Fanuc TP program (LS listing): UP022.LS

/PROG  UP022
/ATTR
OWNER		= MNEDITOR;
COMMENT		= "Soldadura Est.";
PROG_SIZE	= 14814;
CREATE		= DATE 23-07-08  TIME 22:43:52;
MODIFIED	= DATE 24-03-28  TIME 23:41:50;
FILE_NAME	= UP002;
VERSION		= 0;
LINE_COUNT	= 64;
MEMORY_SIZE	= 27222;
PROTECT		= READ_WRITE;
TCD:  STACK_SIZE	= 500,
      TASK_PRIORITY	= 50,
      TIME_SLICE	= 0,
      BUSY_LAMP_OFF	= 0,
      ABORT_REQUEST	= 0,
      PAUSE_REQUEST	= 0;
DEFAULT_GROUP	= 1,1,1,1,*;
CONTROL_CODE	= 00000001 00000000;
/APPL
/MN
   1:  UFRAME_NUM=1 ;
   2:  UTOOL_NUM=2 ;
   3:  PAYLOAD[2] ;
   4:J P[1] 100% CNT0 ACC100 TB    .10sec,P-SPS    ;
      1:  TC_ONLINE (ON) ;
      2:  DO[23]=OFF ;
      3:  TIMER[4]=RESET ;
      4:  TIMER[4]=START ;
      5:  CALL MAKRO050    ;
      6:  !Lib. de Herramientas ;
      7:  DO[80]=ON ;
      8:  DO[79]=ON ;
      9:  DO[78]=OFF ;
     10:  DO[77]=OFF ;
     11:  DO[76]=OFF ;
     12:  DO[75]=ON ;
     13:  DO[73]=OFF ;
     14:  !RLib. de Anticolisiones ;
     15:  DO[41]=ON ;
     16:  DO[42]=ON ;
     17:  DO[43]=ON ;
     18:  DO[44]=ON ;
     19:  DO[45]=ON ;
     20:  DO[46]=ON ;
     21:  !Apagar Pos. Base ;
     22:  DO[15]=OFF ;
     23:  !Robot en Trayectoria ;
     24:  DO[16]=ON ;
     25:  !Basculante en Pos. de Reposo ;
     26:  IF (!DI[842] AND DO[12]),CALL MAKRO072 ;
     27:  WAIT (M[96])    ;
     28:  WAIT (DI[23])    ;
     29:  DO[23]=(ON) ;
     30:  TC_ONLINE (M[1] AND M[30] AND M[31] AND M[34] AND M[95] AND M[96]) ;
       ------ ;
   5:J P[2] 100% CNT100 ACC100 TB   0.00sec,P-SPS    ;
      1:  TC_ONLINE (M[1] AND M[30] AND M[31] AND M[34] AND M[95] AND M[96]) ;
       ------ ;
   6:J P[3] 100% CNT100 ACC100 TB   0.00sec,P-SPS    ;
      1:  TC_ONLINE (M[1] AND M[30] AND M[31] AND M[34] AND M[95] AND M[96]) ;
       ------ ;
   7:J P[4] 100% CNT100 ACC100 TB   0.00sec,P-SPS    ;
      1:  TC_ONLINE (M[1] AND M[30] AND M[31] AND M[34] AND M[95] AND M[96]) ;
       ------ ;
   8:J P[5] 100% CNT100 ACC100 TB   0.00sec,P-SPS    ;
      1:  TC_ONLINE (M[1] AND M[30] AND M[31] AND M[34] AND M[95] AND M[96]) ;
       ------ ;
   9:  !5QA802035B_019_T_PS_0007 ;
  10:  !Punto de Sol. No. 10081 ;
  11:J P[6] 100% CNT0 ACC100 TB    .10sec,P-SPS Offset,PR[11]    ;
      1:  TC_ONLINE (ON) ;
      2:  DO[23]=OFF ;
      3:  WAIT (!DI[16] AND DI[23])    ;
      4:  CALL VW_USER(Basic1,EZSP,Nr1,ProgNr=99, , ,S-Punkt=10081,Fzg_Typ=7,EIN/AUS=ON) ;
      5:  GO[2]=(R[197]+20) ;
      6:  WAIT (!DI[129] OR DI[26])    ;
      7:  CALL MAKRO080    ;
      8:  WAIT (DI[23])    ;
      9:  DO[23]=ON ;
     10:  TC_ONLINE (M[1] AND M[30] AND M[31] AND M[34] AND M[95] AND M[96]) ;
       ------ ;
  12:J P[7] 100% CNT100 ACC100 TB   0.00sec,P-SPS    ;
      1:  TC_ONLINE (M[1] AND M[30] AND M[31] AND M[34] AND M[95] AND M[96]) ;
       ------ ;
  13:  !5QA802035B_019_T_PS_0008 ;
  14:  !Punto de Sol. No. 10082 ;
  15:J P[8] 100% CNT0 ACC100 TB    .10sec,P-SPS Offset,PR[11]    ;
      1:  TC_ONLINE (ON) ;
      2:  DO[23]=OFF ;
      3:  WAIT (!DI[16] AND DI[23])    ;
      4:  CALL VW_USER(Basic1,EZSP,Nr1,ProgNr=99, , ,S-Punkt=10082,Fzg_Typ=7,EIN/AUS=ON) ;
      5:  GO[2]=(R[197]+20) ;
      6:  WAIT (!DI[129] OR DI[26])    ;
      7:  CALL MAKRO080    ;
      8:  WAIT (DI[23])    ;
      9:  DO[23]=ON ;
     10:  TC_ONLINE (M[1] AND M[30] AND M[31] AND M[34] AND M[95] AND M[96]) ;
       ------ ;
  16:  !5QA802035B_019_T_PS_0002 ;
  17:  !Punto de Sol. No. 10083 ;
  18:J P[9] 100% CNT0 ACC100 TB    .10sec,P-SPS Offset,PR[11]    ;
      1:  TC_ONLINE (ON) ;
      2:  DO[23]=OFF ;
      3:  WAIT (!DI[16] AND DI[23])    ;
      4:  CALL VW_USER(Basic1,EZSP,Nr1,ProgNr=99, , ,S-Punkt=10083,Fzg_Typ=7,EIN/AUS=ON) ;
      5:  GO[2]=(R[197]+20) ;
      6:  WAIT (!DI[129] OR DI[26])    ;
      7:  CALL MAKRO080    ;
      8:  WAIT (DI[23])    ;
      9:  DO[23]=ON ;
     10:  TC_ONLINE (M[1] AND M[30] AND M[31] AND M[34] AND M[95] AND M[96]) ;
       ------ ;
  19:  !5QA802035B_019_T_PS_0003 ;
  20:  !Punto de Sol. No. 10084 ;
  21:J P[10] 100% CNT0 ACC100 TB    .10sec,P-SPS Offset,PR[11]    ;
      1:  TC_ONLINE (ON) ;
      2:  DO[23]=OFF ;
      3:  WAIT (!DI[16] AND DI[23])    ;
      4:  CALL VW_USER(Basic1,EZSP,Nr1,ProgNr=99, , ,S-Punkt=10084,Fzg_Typ=7,EIN/AUS=ON) ;
      5:  GO[2]=(R[197]+20) ;
      6:  WAIT (!DI[129] OR DI[26])    ;
      7:  CALL MAKRO080    ;
      8:  WAIT (DI[23])    ;
      9:  DO[23]=ON ;
     10:  TC_ONLINE (M[1] AND M[30] AND M[31] AND M[34] AND M[95] AND M[96]) ;
       ------ ;
  22:  !5QA802035B_019_T_PS_0009 ;
  23:  !Punto de Sol. No. 10085 ;
  24:J P[11] 100% CNT0 ACC100 TB    .10sec,P-SPS Offset,PR[11]    ;
      1:  TC_ONLINE (ON) ;
      2:  DO[23]=OFF ;
      3:  WAIT (!DI[16] AND DI[23])    ;
      4:  CALL VW_USER(Basic1,EZSP,Nr1,ProgNr=99, , ,S-Punkt=10085,Fzg_Typ=7,EIN/AUS=ON) ;
      5:  GO[2]=(R[197]+20) ;
      6:  WAIT (!DI[129] OR DI[26])    ;
      7:  CALL MAKRO080    ;
      8:  WAIT (DI[23])    ;
      9:  DO[23]=ON ;
     10:  TC_ONLINE (M[1] AND M[30] AND M[31] AND M[34] AND M[95] AND M[96]) ;
       ------ ;
  25:J P[12] 100% CNT100 ACC100 TB   0.00sec,P-SPS    ;
      1:  TC_ONLINE (M[1] AND M[30] AND M[31] AND M[34] AND M[95] AND M[96]) ;
       ------ ;
  26:   ;
  27:  !5QA802035B_019_T_PS_0001 ;
  28:  !Punto de Sol. No. 10086 ;
  29:J P[13] 100% CNT0 ACC100 TB    .10sec,P-SPS Offset,PR[11]    ;
      1:  TC_ONLINE (ON) ;
      2:  DO[23]=OFF ;
      3:  WAIT (!DI[16] AND DI[23])    ;
      4:  CALL VW_USER(Basic1,EZSP,Nr1,ProgNr=99, , ,S-Punkt=10086,Fzg_Typ=7,EIN/AUS=ON) ;
      5:  GO[2]=(R[197]+20) ;
      6:  WAIT (!DI[129] OR DI[26])    ;
      7:  CALL MAKRO080    ;
      8:  WAIT (DI[23])    ;
      9:  DO[23]=ON ;
     10:  TC_ONLINE (M[1] AND M[30] AND M[31] AND M[34] AND M[95] AND M[96]) ;
       ------ ;
  30:  !5QA802035B_019_T_PS_0004 ;
  31:  !Punto de Sol. No. 10087 ;
  32:J P[14] 100% CNT0 ACC100 TB    .10sec,P-SPS Offset,PR[11]    ;
      1:  TC_ONLINE (ON) ;
      2:  DO[23]=OFF ;
      3:  WAIT (!DI[16] AND DI[23])    ;
      4:  CALL VW_USER(Basic1,EZSP,Nr1,ProgNr=99, , ,S-Punkt=10087,Fzg_Typ=7,EIN/AUS=ON) ;
      5:  GO[2]=(R[197]+20) ;
      6:  WAIT (!DI[129] OR DI[26])    ;
      7:  CALL MAKRO080    ;
      8:  WAIT (DI[23])    ;
      9:  DO[23]=ON ;
     10:  TC_ONLINE (M[1] AND M[30] AND M[31] AND M[34] AND M[95] AND M[96]) ;
       ------ ;
  33:J P[15] 100% CNT100 ACC100 TB   0.00sec,P-SPS    ;
      1:  TC_ONLINE (M[1] AND M[30] AND M[31] AND M[34] AND M[95] AND M[96]) ;
       ------ ;
  34:  !5QA802035B_055_BN_PS_0001 ;
  35:  !Punto de Sol. No. 10088 ;
  36:J P[16] 100% CNT0 ACC100 TB    .10sec,P-SPS Offset,PR[11]    ;
      1:  TC_ONLINE (ON) ;
      2:  DO[23]=OFF ;
      3:  WAIT (!DI[16] AND DI[23])    ;
      4:  CALL VW_USER(Basic1,EZSP,Nr1,ProgNr=99, , ,S-Punkt=10088,Fzg_Typ=7,EIN/AUS=ON) ;
      5:  GO[2]=(R[197]+20) ;
      6:  WAIT (!DI[129] OR DI[26])    ;
      7:  CALL MAKRO080    ;
      8:  WAIT (DI[23])    ;
      9:  DO[23]=ON ;
     10:  TC_ONLINE (M[1] AND M[30] AND M[31] AND M[34] AND M[95] AND M[96]) ;
       ------ ;
  37:  !5QA802035B_019_T_PS_0005 ;
  38:  !Punto de Sol. No. 10089 ;
  39:J P[17] 100% CNT0 ACC100 TB    .10sec,P-SPS Offset,PR[11]    ;
      1:  TC_ONLINE (ON) ;
      2:  DO[23]=OFF ;
      3:  WAIT (!DI[16] AND DI[23])    ;
      4:  CALL VW_USER(Basic1,EZSP,Nr1,ProgNr=99, , ,S-Punkt=10089,Fzg_Typ=7,EIN/AUS=ON) ;
      5:  GO[2]=(R[197]+20) ;
      6:  WAIT (!DI[129] OR DI[26])    ;
      7:  CALL MAKRO080    ;
      8:  WAIT (DI[23])    ;
      9:  DO[23]=ON ;
     10:  TC_ONLINE (M[1] AND M[30] AND M[31] AND M[34] AND M[95] AND M[96]) ;
       ------ ;
  40:J P[18] 100% CNT100 ACC100 TB   0.00sec,P-SPS    ;
      1:  TC_ONLINE (M[1] AND M[30] AND M[31] AND M[34] AND M[95] AND M[96]) ;
       ------ ;
  41:  !5QA802035B_019_T_PS_0006 ;
  42:  !Punto de Sol. No. 10090 ;
  43:J P[19] 100% CNT0 ACC100 TB    .10sec,P-SPS Offset,PR[11]    ;
      1:  TC_ONLINE (ON) ;
      2:  DO[23]=OFF ;
      3:  WAIT (!DI[16] AND DI[23])    ;
      4:  CALL VW_USER(Basic1,EZSP,Nr1,ProgNr=99, , ,S-Punkt=10090,Fzg_Typ=7,EIN/AUS=ON) ;
      5:  GO[2]=(R[197]+20) ;
      6:  WAIT (!DI[129] OR DI[26])    ;
      7:  CALL MAKRO080    ;
      8:  WAIT (DI[23])    ;
      9:  DO[23]=ON ;
     10:  TC_ONLINE (M[1] AND M[30] AND M[31] AND M[34] AND M[95] AND M[96]) ;
       ------ ;
  44:J P[20] 100% CNT100 ACC100 TB   0.00sec,P-SPS    ;
      1:  TC_ONLINE (M[1] AND M[30] AND M[31] AND M[34] AND M[95] AND M[96]) ;
       ------ ;
  45:J P[21] 100% CNT100 ACC100 TB   0.00sec,P-SPS    ;
      1:  TC_ONLINE (M[1] AND M[30] AND M[31] AND M[34] AND M[95] AND M[96]) ;
       ------ ;
  46:J P[22] 100% CNT100 ACC100 TB   0.00sec,P-SPS    ;
      1:  TC_ONLINE (M[1] AND M[30] AND M[31] AND M[34] AND M[95] AND M[96]) ;
       ------ ;
  47:J P[23] 100% CNT100 ACC100 TB   0.00sec,P-SPS    ;
      1:  TC_ONLINE (M[1] AND M[30] AND M[31] AND M[34] AND M[95] AND M[96]) ;
       ------ ;
  48:J P[24] 100% CNT100 ACC100 TB   0.00sec,P-SPS    ;
      1:  TC_ONLINE (M[1] AND M[30] AND M[31] AND M[34] AND M[95] AND M[96]) ;
       ------ ;
  49:J P[25] 100% CNT100 ACC100 TB   0.00sec,P-SPS    ;
      1:  TC_ONLINE (M[1] AND M[30] AND M[31] AND M[34] AND M[95] AND M[96]) ;
       ------ ;
  50:  !5QA802035B_017_R_PS_0013 ;
  51:  !Punto de Sol. No. 10091 ;
  52:J P[26] 100% CNT0 ACC100 TB    .10sec,P-SPS Offset,PR[11]    ;
      1:  TC_ONLINE (ON) ;
      2:  DO[23]=OFF ;
      3:  WAIT (!DI[16] AND DI[23])    ;
      4:  CALL VW_USER(Basic1,EZSP,Nr1,ProgNr=99, , ,S-Punkt=10091,Fzg_Typ=7,EIN/AUS=ON) ;
      5:  GO[2]=(R[197]+37) ;
      6:  WAIT (!DI[129] OR DI[26])    ;
      7:  CALL MAKRO080    ;
      8:  WAIT (DI[23])    ;
      9:  DO[23]=ON ;
     10:  TC_ONLINE (M[1] AND M[30] AND M[31] AND M[34] AND M[95] AND M[96]) ;
       ------ ;
  53:  !5QA802035B_017_R_PS_0036 ;
  54:  !Punto de Sol. No. 10092 ;
  55:J P[27] 100% CNT0 ACC100 TB    .10sec,P-SPS Offset,PR[11]    ;
      1:  TC_ONLINE (ON) ;
      2:  DO[23]=OFF ;
      3:  WAIT (!DI[16] AND DI[23])    ;
      4:  CALL VW_USER(Basic1,EZSP,Nr1,ProgNr=99, , ,S-Punkt=10092,Fzg_Typ=7,EIN/AUS=ON) ;
      5:  GO[2]=(R[197]+37) ;
      6:  WAIT (!DI[129] OR DI[26])    ;
      7:  CALL MAKRO080    ;
      8:  WAIT (DI[23])    ;
      9:  DO[23]=ON ;
     10:  TC_ONLINE (M[1] AND M[30] AND M[31] AND M[34] AND M[95] AND M[96]) ;
       ------ ;
  56:J P[28] 100% CNT100 ACC100 TB   0.00sec,P-SPS    ;
      1:  TC_ONLINE (M[1] AND M[30] AND M[31] AND M[34] AND M[95] AND M[96]) ;
       ------ ;
  57:  !5QA802035B_017_R_PS_0015 ;
  58:  !Punto de Sol. No. 10093 ;
  59:  !Fin de Trabajo 2 ;
  60:J P[29] 100% CNT0 ACC100 TB    .10sec,P-SPS Offset,PR[11]    ;
      1:  TC_ONLINE (ON) ;
      2:  DO[23]=OFF ;
      3:  WAIT (!DI[16] AND DI[23])    ;
      4:  CALL VW_USER(Basic1,EZSP,Nr1,ProgNr=99, , ,S-Punkt=10093,Fzg_Typ=7,EIN/AUS=ON) ;
      5:  GO[2]=(R[197]+37) ;
      6:  WAIT (!DI[129] OR DI[26])    ;
      7:  CALL MAKRO080    ;
      8:  IF (!DI[145] AND !DI[129]),CALL MAKRO002 ;
      9:  WAIT (DI[23])    ;
     10:  DO[23]=ON ;
     11:  TC_ONLINE (M[1] AND M[30] AND M[31] AND M[34] AND M[95] AND M[96]) ;
       ------ ;
  61:J P[30] 100% CNT100 ACC100 TB   0.00sec,P-SPS    ;
      1:  TC_ONLINE (M[1] AND M[30] AND M[31] AND M[34] AND M[95] AND M[96]) ;
       ------ ;
  62:J P[31] 100% CNT100 ACC100 TB   0.00sec,P-SPS    ;
      1:  TC_ONLINE (M[1] AND M[30] AND M[31] AND M[34] AND M[95] AND M[96]) ;
       ------ ;
  63:J P[32] 100% CNT100 ACC100 TB   0.00sec,P-SPS    ;
      1:  TC_ONLINE (M[1] AND M[30] AND M[31] AND M[34] AND M[95] AND M[96]) ;
       ------ ;
  64:J P[33] 100% CNT0 ACC100 TB    .10sec,P-SPS    ;
      1:  TC_ONLINE (ON) ;
      2:  DO[23]=OFF ;
      3:  TIMER[4]=STOP ;
      4:  WAIT (DI[23])    ;
      5:  CALL VW_USER(Basic1,EZSP,Nr1,ProgNr=31, , ,S-Punkt=31, ,EIN/AUS=1) ;
      6:  DO[23]=ON ;
      7:  TC_ONLINE (M[1] AND M[30] AND M[31] AND M[34] AND M[95] AND M[96]) ;
       ------ ;
/POS
P[1]{
   GP1:
	UF : 1, UT : 2,		CONFIG : 'N U T, 0, 0, 0',
	RX =   -96.676  mm,	RY = -1778.617  mm,	RZ =  -961.637  mm,
	RW =   124.259 deg,	RP =    62.839 deg,	RR =  -172.987 deg
   GP2:
	UF : 1, UT : 2,
	J1=   100.000  mm
   GP3:
	UF : 1, UT : 2,
	J1=     0.000  mm
   GP4:
	UF : 1, UT : 2,
	J1=     0.000  mm
};
P[2]{
   GP1:
	UF : 1, UT : 2,		CONFIG : 'N U T, 0, 0, 0',
	RX =   399.675  mm,	RY = -1124.385  mm,	RZ =  -655.908  mm,
	RW =    82.166 deg,	RP =    59.374 deg,	RR =  -158.331 deg
   GP2:
	UF : 1, UT : 2,
	J1=   110.000  mm
   GP3:
	UF : 1, UT : 2,
	J1=     0.000  mm
   GP4:
	UF : 1, UT : 2,
	J1=     0.000  mm
};
P[3]{
   GP1:
	UF : 1, UT : 2,		CONFIG : 'F U T, 0, 0, 0',
	RX =   288.903  mm,	RY =  -470.311  mm,	RZ =   232.156  mm,
	RW =   126.074 deg,	RP =     7.960 deg,	RR =   -89.771 deg
   GP2:
	UF : 1, UT : 2,
	J1=   110.000  mm
   GP3:
	UF : 1, UT : 2,
	J1=     0.000  mm
   GP4:
	UF : 1, UT : 2,
	J1=     0.000  mm
};
P[4]{
   GP1:
	UF : 1, UT : 2,		CONFIG : 'F U T, 0, 0, 0',
	RX =   188.860  mm,	RY =  -448.835  mm,	RZ =   155.340  mm,
	RW =   123.074 deg,	RP =     7.960 deg,	RR =   -89.771 deg
   GP2:
	UF : 1, UT : 2,
	J1=    60.000  mm
   GP3:
	UF : 1, UT : 2,
	J1=     0.000  mm
   GP4:
	UF : 1, UT : 2,
	J1=     0.000  mm
};
P[5]{
   GP1:
	UF : 1, UT : 2,		CONFIG : 'F U T, 0, 0, 0',
	RX =   147.239  mm,	RY =  -450.492  mm,	RZ =   130.708  mm,
	RW =   123.075 deg,	RP =     7.960 deg,	RR =   -89.771 deg
   GP2:
	UF : 1, UT : 2,
	J1=    60.000  mm
   GP3:
	UF : 1, UT : 2,
	J1=     0.000  mm
   GP4:
	UF : 1, UT : 2,
	J1=     0.000  mm
};
P[6]{
   GP1:
	UF : 1, UT : 2,		CONFIG : 'F U T, 0, 0, 0',
	RX =   151.493  mm,	RY =  -456.934  mm,	RZ =   130.703  mm,
	RW =   123.000 deg,	RP =     7.582 deg,	RR =   -90.159 deg
   GP2:
	UF : 1, UT : 2,
	J1=    24.000  mm
   GP3:
	UF : 1, UT : 2,
	J1=     0.000  mm
   GP4:
	UF : 1, UT : 2,
	J1=     0.000  mm
};
P[7]{
   GP1:
	UF : 1, UT : 2,		CONFIG : 'F U T, 0, 0, 0',
	RX =   153.908  mm,	RY =  -449.432  mm,	RZ =    94.568  mm,
	RW =   125.975 deg,	RP =     7.963 deg,	RR =   -90.511 deg
   GP2:
	UF : 1, UT : 2,
	J1=    25.353  mm
   GP3:
	UF : 1, UT : 2,
	J1=     0.000  mm
   GP4:
	UF : 1, UT : 2,
	J1=     0.000  mm
};
P[8]{
   GP1:
	UF : 1, UT : 2,		CONFIG : 'F U T, 0, 0, 0',
	RX =   153.849  mm,	RY =  -452.627  mm,	RZ =    94.116  mm,
	RW =   126.038 deg,	RP =     8.562 deg,	RR =   -90.071 deg
   GP2:
	UF : 1, UT : 2,
	J1=    24.000  mm
   GP3:
	UF : 1, UT : 2,
	J1=     0.000  mm
   GP4:
	UF : 1, UT : 2,
	J1=     0.000  mm
};
P[9]{
   GP1:
	UF : 1, UT : 2,		CONFIG : 'F U T, 0, 0, 0',
	RX =   133.821  mm,	RY =  -449.815  mm,	RZ =    70.970  mm,
	RW =   125.880 deg,	RP =     8.211 deg,	RR =   -91.003 deg
   GP2:
	UF : 1, UT : 2,
	J1=    24.000  mm
   GP3:
	UF : 1, UT : 2,
	J1=     0.000  mm
   GP4:
	UF : 1, UT : 2,
	J1=     0.000  mm
};
P[10]{
   GP1:
	UF : 1, UT : 2,		CONFIG : 'F U T, 0, 0, 0',
	RX =   106.033  mm,	RY =  -453.176  mm,	RZ =    90.592  mm,
	RW =   127.134 deg,	RP =     8.757 deg,	RR =   -83.385 deg
   GP2:
	UF : 1, UT : 2,
	J1=    24.000  mm
   GP3:
	UF : 1, UT : 2,
	J1=     0.000  mm
   GP4:
	UF : 1, UT : 2,
	J1=     0.000  mm
};
P[11]{
   GP1:
	UF : 1, UT : 2,		CONFIG : 'F U T, 0, 0, 0',
	RX =   122.760  mm,	RY =  -455.458  mm,	RZ =   112.228  mm,
	RW =   127.134 deg,	RP =     8.757 deg,	RR =   -83.385 deg
   GP2:
	UF : 1, UT : 2,
	J1=    18.400  mm
   GP3:
	UF : 1, UT : 2,
	J1=     0.000  mm
   GP4:
	UF : 1, UT : 2,
	J1=     0.000  mm
};
P[12]{
   GP1:
	UF : 1, UT : 2,		CONFIG : 'F U T, 0, 0, 0',
	RX =   118.146  mm,	RY =  -455.286  mm,	RZ =   115.913  mm,
	RW =   125.582 deg,	RP =     8.263 deg,	RR =   -83.694 deg
   GP2:
	UF : 1, UT : 2,
	J1=    27.608  mm
   GP3:
	UF : 1, UT : 2,
	J1=     0.000  mm
   GP4:
	UF : 1, UT : 2,
	J1=     0.000  mm
};
P[13]{
   GP1:
	UF : 1, UT : 2,		CONFIG : 'F U T, 0, 0, 0',
	RX =    99.026  mm,	RY =  -459.413  mm,	RZ =   108.502  mm,
	RW =   112.126 deg,	RP =     7.968 deg,	RR =   -84.170 deg
   GP2:
	UF : 1, UT : 2,
	J1=    24.000  mm
   GP3:
	UF : 1, UT : 2,
	J1=     0.000  mm
   GP4:
	UF : 1, UT : 2,
	J1=     0.000  mm
};
P[14]{
   GP1:
	UF : 1, UT : 2,		CONFIG : 'F U T, 0, 0, 0',
	RX =    73.087  mm,	RY =  -462.671  mm,	RZ =   109.873  mm,
	RW =   106.997 deg,	RP =     6.853 deg,	RR =   -79.767 deg
   GP2:
	UF : 1, UT : 2,
	J1=    24.000  mm
   GP3:
	UF : 1, UT : 2,
	J1=     0.000  mm
   GP4:
	UF : 1, UT : 2,
	J1=     0.000  mm
};
P[15]{
   GP1:
	UF : 1, UT : 2,		CONFIG : 'F U T, 0, 0, 0',
	RX =    61.641  mm,	RY =  -463.963  mm,	RZ =   132.664  mm,
	RW =    95.632 deg,	RP =     5.204 deg,	RR =   -83.060 deg
   GP2:
	UF : 1, UT : 2,
	J1=    30.000  mm
   GP3:
	UF : 1, UT : 2,
	J1=     0.000  mm
   GP4:
	UF : 1, UT : 2,
	J1=     0.000  mm
};
P[16]{
   GP1:
	UF : 1, UT : 2,		CONFIG : 'F U T, 0, 0, 0',
	RX =    57.906  mm,	RY =  -466.475  mm,	RZ =   139.419  mm,
	RW =    95.518 deg,	RP =     5.325 deg,	RR =   -84.305 deg
   GP2:
	UF : 1, UT : 2,
	J1=    24.000  mm
   GP3:
	UF : 1, UT : 2,
	J1=     0.000  mm
   GP4:
	UF : 1, UT : 2,
	J1=     0.000  mm
};
P[17]{
   GP1:
	UF : 1, UT : 2,		CONFIG : 'F U T, 0, 0, 0',
	RX =    83.720  mm,	RY =  -463.217  mm,	RZ =   129.706  mm,
	RW =   103.991 deg,	RP =     8.585 deg,	RR =   -82.834 deg
   GP2:
	UF : 1, UT : 2,
	J1=    24.000  mm
   GP3:
	UF : 1, UT : 2,
	J1=     0.000  mm
   GP4:
	UF : 1, UT : 2,
	J1=     0.000  mm
};
P[18]{
   GP1:
	UF : 1, UT : 2,		CONFIG : 'F U T, 0, 0, 0',
	RX =    83.058  mm,	RY =  -459.334  mm,	RZ =   130.270  mm,
	RW =   104.348 deg,	RP =     7.966 deg,	RR =   -80.363 deg
   GP2:
	UF : 1, UT : 2,
	J1=    30.000  mm
   GP3:
	UF : 1, UT : 2,
	J1=     0.000  mm
   GP4:
	UF : 1, UT : 2,
	J1=     0.000  mm
};
P[19]{
   GP1:
	UF : 1, UT : 2,		CONFIG : 'F U T, 0, 0, 0',
	RX =   128.594  mm,	RY =  -459.074  mm,	RZ =   132.498  mm,
	RW =   110.390 deg,	RP =     8.524 deg,	RR =   -87.108 deg
   GP2:
	UF : 1, UT : 2,
	J1=    24.000  mm
   GP3:
	UF : 1, UT : 2,
	J1=     0.000  mm
   GP4:
	UF : 1, UT : 2,
	J1=     0.000  mm
};
P[20]{
   GP1:
	UF : 1, UT : 2,		CONFIG : 'F U T, 0, 0, 0',
	RX =   125.268  mm,	RY =  -454.795  mm,	RZ =   133.527  mm,
	RW =   110.548 deg,	RP =     7.953 deg,	RR =   -86.047 deg
   GP2:
	UF : 1, UT : 2,
	J1=   110.000  mm
   GP3:
	UF : 1, UT : 2,
	J1=     0.000  mm
   GP4:
	UF : 1, UT : 2,
	J1=     0.000  mm
};
P[21]{
   GP1:
	UF : 1, UT : 2,		CONFIG : 'F U T, 0, 0, 0',
	RX =   158.073  mm,	RY =  -447.089  mm,	RZ =   130.598  mm,
	RW =   117.548 deg,	RP =     7.953 deg,	RR =   -86.047 deg
   GP2:
	UF : 1, UT : 2,
	J1=   110.000  mm
   GP3:
	UF : 1, UT : 2,
	J1=     0.000  mm
   GP4:
	UF : 1, UT : 2,
	J1=     0.000  mm
};
P[22]{
   GP1:
	UF : 1, UT : 2,		CONFIG : 'F U T, 0, 0, 0',
	RX =   161.685  mm,	RY =  -448.970  mm,	RZ =   131.093  mm,
	RW =   127.548 deg,	RP =     7.953 deg,	RR =   -86.047 deg
   GP2:
	UF : 1, UT : 2,
	J1=   110.000  mm
   GP3:
	UF : 1, UT : 2,
	J1=     0.000  mm
   GP4:
	UF : 1, UT : 2,
	J1=     0.000  mm
};
P[23]{
   GP1:
	UF : 1, UT : 2,		CONFIG : 'F U T, 0, 0, 0',
	RX =   221.390  mm,	RY =  -458.710  mm,	RZ =   186.318  mm,
	RW =   124.547 deg,	RP =     7.953 deg,	RR =   -86.047 deg
   GP2:
	UF : 1, UT : 2,
	J1=   110.000  mm
   GP3:
	UF : 1, UT : 2,
	J1=     0.000  mm
   GP4:
	UF : 1, UT : 2,
	J1=     0.000  mm
};
P[24]{
   GP1:
	UF : 1, UT : 2,		CONFIG : 'F U T, 0, 0, 0',
	RX =   183.432  mm,	RY =  -464.818  mm,	RZ =   254.976  mm,
	RW =   141.048 deg,	RP =    10.000 deg,	RR =   -87.700 deg
   GP2:
	UF : 1, UT : 2,
	J1=    60.000  mm
   GP3:
	UF : 1, UT : 2,
	J1=     0.000  mm
   GP4:
	UF : 1, UT : 2,
	J1=     0.000  mm
};
P[25]{
   GP1:
	UF : 1, UT : 2,		CONFIG : 'F U T, 0, 0, 0',
	RX =   142.455  mm,	RY =  -476.613  mm,	RZ =   238.754  mm,
	RW =   148.668 deg,	RP =    10.183 deg,	RR =   -87.938 deg
   GP2:
	UF : 1, UT : 2,
	J1=    30.000  mm
   GP3:
	UF : 1, UT : 2,
	J1=     0.000  mm
   GP4:
	UF : 1, UT : 2,
	J1=     0.000  mm
};
P[26]{
   GP1:
	UF : 1, UT : 2,		CONFIG : 'F U T, 0, 0, 0',
	RX =   141.357  mm,	RY =  -475.116  mm,	RZ =   214.449  mm,
	RW =   148.129 deg,	RP =     7.165 deg,	RR =   -89.090 deg
   GP2:
	UF : 1, UT : 2,
	J1=    21.300  mm
   GP3:
	UF : 1, UT : 2,
	J1=     0.000  mm
   GP4:
	UF : 1, UT : 2,
	J1=     0.000  mm
};
P[27]{
   GP1:
	UF : 1, UT : 2,		CONFIG : 'F U T, 0, 0, 0',
	RX =   118.024  mm,	RY =  -476.373  mm,	RZ =   215.669  mm,
	RW =   149.383 deg,	RP =     9.640 deg,	RR =   -91.683 deg
   GP2:
	UF : 1, UT : 2,
	J1=    12.800  mm
   GP3:
	UF : 1, UT : 2,
	J1=     0.000  mm
   GP4:
	UF : 1, UT : 2,
	J1=     0.000  mm
};
P[28]{
   GP1:
	UF : 1, UT : 2,		CONFIG : 'F U T, 0, 0, 0',
	RX =   131.388  mm,	RY =  -471.170  mm,	RZ =   230.494  mm,
	RW =   149.074 deg,	RP =    10.000 deg,	RR =   -87.700 deg
   GP2:
	UF : 1, UT : 2,
	J1=    30.000  mm
   GP3:
	UF : 1, UT : 2,
	J1=     0.000  mm
   GP4:
	UF : 1, UT : 2,
	J1=     0.000  mm
};
P[29]{
   GP1:
	UF : 1, UT : 2,		CONFIG : 'F U T, 0, 0, 0',
	RX =    67.750  mm,	RY =  -474.998  mm,	RZ =   234.118  mm,
	RW =   137.625 deg,	RP =     9.670 deg,	RR =   -99.963 deg
   GP2:
	UF : 1, UT : 2,
	J1=    20.300  mm
   GP3:
	UF : 1, UT : 2,
	J1=     0.000  mm
   GP4:
	UF : 1, UT : 2,
	J1=     0.000  mm
};
P[30]{
   GP1:
	UF : 1, UT : 2,		CONFIG : 'F U T, 0, 0, 0',
	RX =    71.063  mm,	RY =  -462.382  mm,	RZ =   241.583  mm,
	RW =   143.581 deg,	RP =    10.000 deg,	RR =   -87.700 deg
   GP2:
	UF : 1, UT : 2,
	J1=   110.000  mm
   GP3:
	UF : 1, UT : 2,
	J1=     0.000  mm
   GP4:
	UF : 1, UT : 2,
	J1=     0.000  mm
};
P[31]{
   GP1:
	UF : 1, UT : 2,		CONFIG : 'F U T, 0, 0, 0',
	RX =   129.166  mm,	RY =  -484.273  mm,	RZ =   308.532  mm,
	RW =   141.048 deg,	RP =    10.000 deg,	RR =   -87.700 deg
   GP2:
	UF : 1, UT : 2,
	J1=   110.000  mm
   GP3:
	UF : 1, UT : 2,
	J1=     0.000  mm
   GP4:
	UF : 1, UT : 2,
	J1=     0.000  mm
};
P[32]{
   GP1:
	UF : 1, UT : 2,		CONFIG : 'F U T, 0, 0, 0',
	RX =   343.407  mm,	RY =  -832.324  mm,	RZ =   497.055  mm,
	RW =   141.047 deg,	RP =    10.000 deg,	RR =   -87.701 deg
   GP2:
	UF : 1, UT : 2,
	J1=   110.000  mm
   GP3:
	UF : 1, UT : 2,
	J1=     0.000  mm
   GP4:
	UF : 1, UT : 2,
	J1=     0.000  mm
};
P[33]{
   GP1:
	UF : 1, UT : 2,		CONFIG : 'N U T, 0, 0, 0',
	RX =   -96.677  mm,	RY = -1778.618  mm,	RZ =  -961.636  mm,
	RW =   124.259 deg,	RP =    62.839 deg,	RR =  -172.987 deg
   GP2:
	UF : 1, UT : 2,
	J1=   100.000  mm
   GP3:
	UF : 1, UT : 2,
	J1=     0.000  mm
   GP4:
	UF : 1, UT : 2,
	J1=     0.000  mm
};
/END
